Fanuc KAREL source: kx00032.KL

-- PROVISIONAL review KL for V770-1; original PC SHA256 8fce5f46047be16b6aa1acea95ba738a54815a626f7da3f11f314f69c6acc03f
-- Incomplete behavior may be omitted. Consult companion uncertainty JSON. Do not deploy.
PROGRAM KX00032
%NOLOCKGROUP
VAR
  I : INTEGER
  J : INTEGER
  B : BOOLEAN
  F : FILE
  S : STRING[80]
-- UNRESOLVED_DECL P type=000102
BEGIN
  -- UNRESOLVED_PC offsets 5-12; opcodes 9D,23
  -- UNRESOLVED_PC offsets 17-21; opcodes 7F
END KX00032
